FUNCTION_BLOCK FB_Stromzaehler_Gebaeude
VAR_INPUT
	Telegramm	: ARRAY[1..cMBUS_MaxTelegrams] OF ST_MBus_Data2;
END_VAR
VAR_IN_OUT
	Zustand		: ST_SZ_Zustand;
END_VAR
VAR
	Leistungsberechnung			: FB_ABB_Lesen;
END_VAR
VAR // added by the converter: edge detectors and wires of the graphical bodies
    _w1 : ANY;
END_VAR

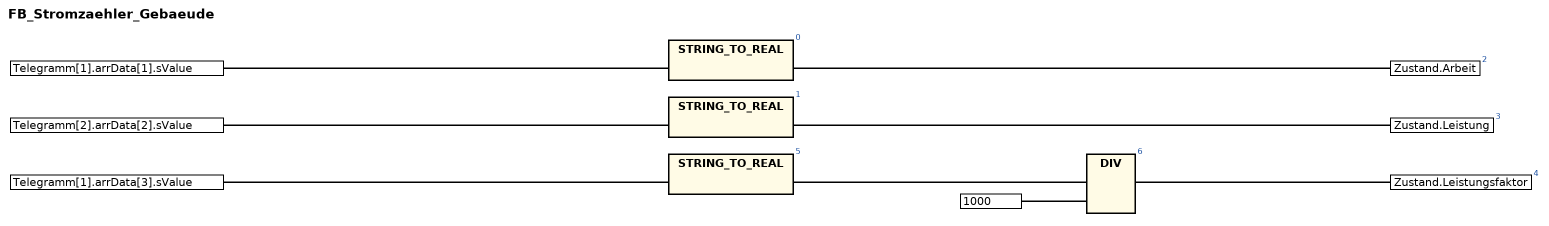
Zustand.Arbeit := STRING_TO_REAL(Telegramm[1].arrData[1].sValue);
Zustand.Leistung := STRING_TO_REAL(Telegramm[2].arrData[2].sValue);
Zustand.Leistungsfaktor := _w1;
_w1 := STRING_TO_REAL(Telegramm[1].arrData[3].sValue) / 1000;

END_FUNCTION_BLOCK

(* stored: Version 1.1.0.1, ProductVersion 3.1.4024.9
   POU FB_Stromzaehler_Gebaeude: Id {4e484e2c-6944-4f0a-8c38-949683e4612a}, SpecialFunc None *)
